FUNCTION_BLOCK FB_Boiler EXTENDS FB_PackML_BaseModule IMPLEMENTS I_Boiler
VAR
	// Interfaces
	ipHeatingElement 	:	I_HeatingElement;
	ipTempSensor 		: 	I_TempSensor;
	
	// FBs
	Sim_Heater 					: FB_SimulatedHeater;
	Sim_TempSensor 				: FB_SimulatedTempSensor;
	
	// Local Variables
	_TemperatureSetpoint	: LREAL;
	_Heating				: BOOL;
	_SimulateComponents: BOOL;
END_VAR

PROPERTY CurrentTemp : LREAL
GET
IF ipTempSensor <> 0 THEN
	CurrentTemp := ipTempSensor.Temp;
END_IF
END_GET
END_PROPERTY

//{warning 'Add method implementation '}
METHOD CyclicLogic
VAR
END_VAR
IF _SimulateComponents THEN
	ipHeatingElement := Sim_Heater;
	ipTempSensor := Sim_TempSensor;
	ipTempSensor.SimulatedHeatingElement := ipHeatingElement;
END_IF

IF ipTempSensor <> 0 AND ipHeatingElement <> 0 THEN
	IF ipTempSensor.Temp < _TemperatureSetpoint THEN
		ipHeatingElement.PowerOn();
		_Heating := TRUE;
	ELSE
		ipHeatingElement.PowerOff();
		_Heating := FALSE;
	END_IF
	
	ipTempSensor.CyclicLogic();
	ipHeatingElement.CyclicLogic();
END_IF
END_METHOD

{warning 'Add method implementation '}
METHOD Disable : BOOL
END_METHOD

{warning 'Add method implementation '}
METHOD Enable : BOOL
END_METHOD

PROPERTY Heating : BOOL
GET
Heating := _Heating;
END_GET
END_PROPERTY

{warning 'Add property implementation'}
PROPERTY SetpointMet : BOOL
GET
END_GET
END_PROPERTY

PROPERTY SimulateComponents : BOOL
GET
SimulateComponents := _SimulateComponents;
END_GET
SET
_SimulateComponents := SimulateComponents;
END_SET
END_PROPERTY

{warning 'Add property implementation'}
PROPERTY TemperatureSetpoint : LREAL
GET
END_GET
SET
END_SET
END_PROPERTY

END_FUNCTION_BLOCK

(* stored: Version 1.1.0.1
   POU FB_Boiler: Id {34b3672c-408e-44c2-8295-16ea1aa1e18a}, SpecialFunc None
   Property CurrentTemp: Id {db351b7c-035a-4942-ab59-70a6cc37df24}
   Get Get: Id {40696634-8714-4025-a9f1-f0fc293b5eb6}
   Method CyclicLogic: Id {5091d7f9-b204-46ec-936d-18b529bb496d}
   Method Disable: Id {f60e66fc-af66-444e-adf7-cb5c9addbc75}
   Method Enable: Id {cdb83fee-485f-4db6-b4ca-82ec4e83e942}
   Property Heating: Id {18430da4-247c-4dc2-b3d6-d4cab408d20e}
   Get Get: Id {31816ab3-92e3-4a00-a4a8-55583b54bc7c}
   Property SetpointMet: Id {ab534255-e398-44fe-ac3f-14ee4188a5b0}
   Get Get: Id {cb0dd34b-d7a4-4a3b-b956-35c089498b32}
   Property SimulateComponents: Id {1a92ceb2-72ac-4d85-bfb7-6c3a863a35b0}
   Get Get: Id {c72b9250-f358-40bb-951c-d11a8a2bd16a}
   Set Set: Id {6ae34b39-3fba-45b4-bdf7-cbc9dc5e80c5}
   Property TemperatureSetpoint: Id {9c79338d-b453-42c1-a2fe-92ffdeaf30a0}
   Get Get: Id {fad31b38-fa26-4abb-83ae-0df8a9d07515}
   Set Set: Id {3fff3071-2f7a-43de-9b8c-508fbc602e15} *)
